TYPE AxesSetPositionProcessArgs :
STRUCT
	///New position to be taken over by the axis
	value: LREAL;
END_STRUCT
END_TYPE

(* stored: Version 1.1.0.1, ProductVersion 3.1.4019.2
   DUT AxesSetPositionProcessArgs: Id {8ace42a7-e0e1-4854-81c9-8c5cb1667301} *)
